FUNCTION_BLOCK Q_ChildLocation (* Command change child location ( Part 6 - F.14 ) *)
  (* Standard: ISO 11783-6; Description: Copyright (c) 2022 HR Agrartechnik GmbH This program and the accompanying materials are made available under the terms of the Eclipse Public License 2.0 which is available at https://www.eclipse.org/legal/epl-2.0/ SPDX-License-Identifier: EPL-2.0 see Description Tab *)
  (* Version 1.0, 2022-07-08, Franz Höpfinger, HR Agrartechnik GmbH *)
  PACKAGE isobus::UT::Q;
  IMPORT eclipse4diac::core::TypeHash;
  IMPORT isobus::UT::Q::IDs::ID_NULL;
  (* Documentation:
  Command change child location ( Part 6 - F.14 )
   The Change Child Location command is used to change the relative position of an object.
   param[in] {objectID, uint16_t}
   Object ID
   param[in] {parentObjectID, uint16_t}
   Parent object ID
   param[in] {relativeXPositionChange, uint8_t}
   Relative change in x position (interpreted as signed!)
   param[in] {relativeYPositionChange, uint8_t}
   Relative change in y position (interpreted as signed!)
   Return Values: 
   int16_t
    - VT_E_NO_ERR (0) - OK
   - VT_E_OVERFLOW (-6) - buffer overflow
   - VT_E_NOACT (-8) - Command not possible in current state
   - VT_E_NO_INSTANCE (-21) - No VT client available
   - VT_E_ISO_INSTANCE_INVALID (-129) - Identifier for instance (connection) invalid
   - VT_E_NOT_ALIVE (-130) - Identifier for instance valid, but VT Dead.
  *)
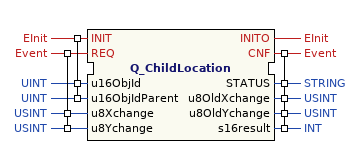
  EVENT_INPUT
    INIT : EInit WITH u16ObjId, u16ObjIdParent; (* Service Initialization *)
    REQ WITH u8Xchange, u8Ychange; (* Service Request *)
  END_EVENT
  EVENT_OUTPUT
    INITO : EInit; (* Initialization Confirm *)
    CNF WITH STATUS, u8OldYchange, u8OldXchange, s16result; (* Confirmation of Requested Service *)
  END_EVENT
  VAR_INPUT
    u16ObjId : UINT := ID_NULL; (* Object ID *)
    u16ObjIdParent : UINT := ID_NULL; (* Parent object ID *)
    u8Xchange : USINT; (* Relative change in x position (interpreted as signed!) *)
    u8Ychange : USINT; (* Relative change in y position (interpreted as signed!) *)
  END_VAR
  VAR_OUTPUT
    STATUS : STRING; (* Service Status *)
    u8OldXchange : USINT; (* Old relative change in x position (interpreted as signed!) *)
    u8OldYchange : USINT; (* Old relative change in y position (interpreted as signed!) *)
    s16result : INT; (* retval see description *)
  END_VAR
END_FUNCTION_BLOCK
